{attribute 'qualified_only'}
VAR_GLOBAL
	Contador : INT := 50;
	SetpointVelocidade : REAL := 20;
END_VAR

(* stored: Version 1.1.0.1
   GVL GVL: Id {dd41b6df-90ea-4f09-bfac-4f3747178658} *)
